FUNCTION_BLOCK PLCnextAXLSEDI16 (* Service Interface Function Block Type *)
  (* Standard: 61499-2; Description: Copyright (c) 2022 Peirlberger Juergen This program and the accompanying materials are made available under the terms of the Eclipse Public License 2.0 which is available at https://www.eclipse.org/legal/epl-2.0/ SPDX-License-Identifier: EPL-2.0 *)
  (* Version 3.0, 2025-04-14, Patrick Aigner, changed package *)
  (* Version 1.0, 2022-04-07, Peirlberger Juergen *)
  PACKAGE eclipse4diac::io::plcnext;
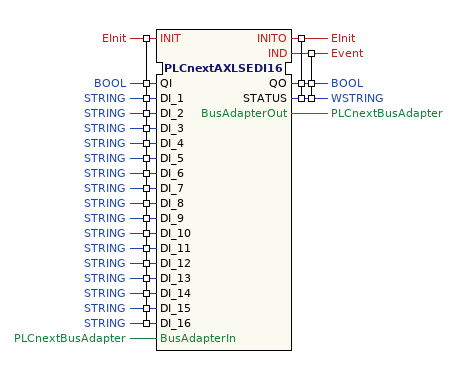
  EVENT_INPUT
    INIT : EInit WITH QI, DI_1, DI_2, DI_3, DI_4, DI_5, DI_6, DI_7, DI_8, DI_9, DI_10, DI_11, DI_12, DI_13, DI_14, DI_15, DI_16; (* Service Initialization *)
  END_EVENT
  EVENT_OUTPUT
    INITO : EInit WITH QO, STATUS; (* Initialization Confirm *)
    IND WITH QO, STATUS; (* Indication from Resource *)
  END_EVENT
  VAR_INPUT
    QI : BOOL; (* Event Input Qualifier *)
    DI_1 : STRING; (* Digital Input *)
    DI_2 : STRING; (* Digital Input *)
    DI_3 : STRING; (* Digital Input *)
    DI_4 : STRING; (* Digital Input *)
    DI_5 : STRING; (* Digital Input *)
    DI_6 : STRING; (* Digital Input *)
    DI_7 : STRING; (* Digital Input *)
    DI_8 : STRING; (* Digital Input *)
    DI_9 : STRING; (* Digital Input *)
    DI_10 : STRING; (* Digital Input *)
    DI_11 : STRING; (* Digital Input *)
    DI_12 : STRING; (* Digital Input *)
    DI_13 : STRING; (* Digital Input *)
    DI_14 : STRING; (* Digital Input *)
    DI_15 : STRING; (* Digital Input *)
    DI_16 : STRING; (* Digital Input *)
  END_VAR
  VAR_OUTPUT
    QO : BOOL; (* Event Output Qualifier *)
    STATUS : WSTRING; (* Service Status *)
  END_VAR
  SOCKETS
    BusAdapterIn : eclipse4diac::io::plcnext::PLCnextBusAdapter;
  END_SOCKETS
  PLUGS
    BusAdapterOut : eclipse4diac::io::plcnext::PLCnextBusAdapter;
  END_PLUGS
END_FUNCTION_BLOCK
